TEXTLIST StationAckMode_txt
  0 = 'Time'
  1 = 'External Ack'
   = ''
END_TEXTLIST

(* stored: Version 1.1.0.1, ProductVersion 3.1.4024.11
   TextList StationAckMode_txt: Id {9c52a165-aebd-422a-afbd-e6623bb53781} *)
